// TIA Portal V20 export
FUNCTION "fc_2" : Void   // FC1, LAD
{ S7_Optimized_Access := 'TRUE' }
// stored: SetENOAutomatically false
   VAR_TEMP
      ton_attivato : Bool;
      tof_attivato : Bool;
      conto_ctu_finito : Bool;
      reset_ctu : Bool;
      attiva_ton : Bool;
      attiva_tof : Bool;
      conta_ctu : Bool;
   END_VAR
BEGIN

REGION Network 1: ton
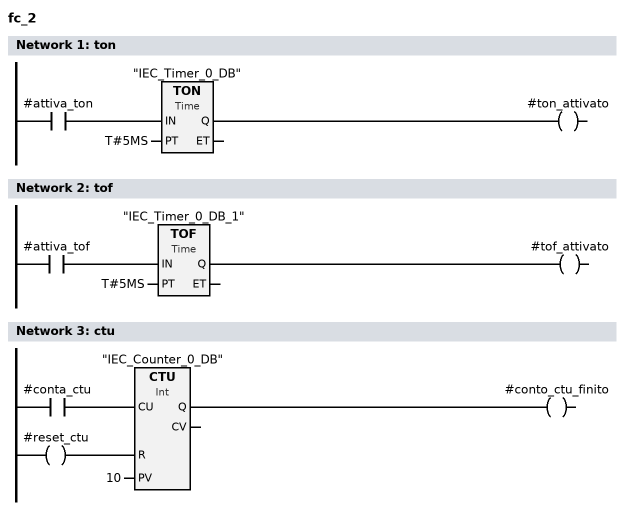
   RUNG wire#powerrail
      Contact( #attiva_ton )
      { S7_Templates := "time_type := Time" } "IEC_Timer_0_DB".TON(pt := T#5MS, et =>)
      Coil( #ton_attivato )
   END_RUNG
   // the same network as SCL:
   "IEC_Timer_0_DB".TON(IN := #attiva_ton, PT := T#5MS);
   #ton_attivato := "IEC_Timer_0_DB".Q;
END_REGION

REGION Network 2: tof
   RUNG wire#powerrail
      Contact( #attiva_tof )
      { S7_Templates := "time_type := Time" } "IEC_Timer_0_DB_1".TOF(pt := T#5MS, et =>)
      Coil( #tof_attivato )
   END_RUNG
   // the same network as SCL:
   "IEC_Timer_0_DB_1".TOF(IN := #attiva_tof, PT := T#5MS);
   #tof_attivato := "IEC_Timer_0_DB_1".Q;
END_REGION

REGION Network 3: ctu
   RUNG wire#powerrail
      Contact( #conta_ctu )
      { S7_Templates := "value_type := Int" } "IEC_Counter_0_DB".CTU(r := wire#w1, pv := 10, cv =>)
      Coil( #conto_ctu_finito )
   END_RUNG
   RUNG wire#powerrail
      Coil( #reset_ctu )
   END_RUNG wire#w1
   // the same network as SCL:
   #reset_ctu := TRUE;
   "IEC_Counter_0_DB".CTU(CU := #conta_ctu, R := TRUE, PV := 10);
   #conto_ctu_finito := "IEC_Counter_0_DB".Q;
END_REGION
END_FUNCTION
